INTERFACE I_V1_Virtual_Input_Source EXTENDS I_VirtualInputSource

PROPERTY nV1_tMlCalculation : UDINT
GET
END_GET
END_PROPERTY

PROPERTY nV1_nUnitsProduced : ULINT
GET
END_GET
END_PROPERTY

PROPERTY nV1_nDefectiveUnits : ULINT
GET
END_GET
END_PROPERTY

PROPERTY nV1_nState : UINT
GET
END_GET
END_PROPERTY

END_INTERFACE

(* stored: Itf I_V1_Virtual_Input_Source: Id 661604dc-1a99-4680-8897-20e6bf6d6450
   Property nV1_tMlCalculation: Id f0d3ac12-416b-4da2-84b0-693194305e3d
   Get Get: Id f90f10c2-0d23-46cf-94e5-7e5c28126901
   Property nV1_nUnitsProduced: Id dad5736f-eb78-4bbc-b8eb-6a583522b7c7
   Get Get: Id d614fc1e-5014-404e-a2cd-abd5bfcc066b
   Property nV1_nDefectiveUnits: Id 0ed0c310-7a83-43c8-988e-de007ff4b487
   Get Get: Id ce546a8d-7f26-4509-958c-492720c3e1d0
   Property nV1_nState: Id 09e98601-c401-4f65-8fea-6ef7c0826bda
   Get Get: Id 435f2981-d226-422e-b3a5-e6082188cfe0 *)
